{attribute 'GeneratedUsingTerminal: EP1312-0001-0016'}
{attribute addProperty BoxType "EP1312-0001-0016"}
{attribute addProperty Id "EtcSlaveTerminalBaseInfoDataAT %I*InfoData_6F19DB2B2"}
{attribute addProperty CRC "2874840167"}
{attribute addProperty Size "2"}
TYPE EP1312_AB5A9467 EXTENDS EtcSlaveTerminalBase :
STRUCT
	{attribute addProperty Name "InfoData"}
	InfoData : InfoData_6F19DB2B;
END_STRUCT
END_TYPE

(* stored: Version 1.2.0.0, ProductVersion 3.1.4024.9
   DUT EP1312_AB5A9467: Id {c51c5abe-8d5c-4c3a-94d3-a8d955a39957} *)
